Staubli VAL3: ex11.pjx

Parameters version=s7.4 stackSize=5000 millimeterUnit=true
Program file=exo11.pgx
Program file=start.pgx
Program file=stop.pgx
Data file=ex11.dtx
